TYPE "UDT_ZC_RECETA_CIP_ESTERIL"
VERSION : 0.1
   STRUCT
      TiempoEmpujeADestino : Int;   // ESTERILIZACIÓN. Tiempo de empuje a destino
      TiempoMaxVaciadoDestino : Int;   // ESTERILIZACIÓN. Tiempo Max vaciado destino
      TiempoEmpujeDestinoACIP : Int;   // ESTERILIZACIÓN. Tiempoi empuje desde equipo a CIP
      TiempoMaxEsterilizacion : Int;   // ESTERILIZACIÓN. Tiempo Maximo Enjuague
      TiempoEsterilizacionConConductividad : Int;   // ESTERILIZACIÓN. Tiempo enjuague con conductividad
      ReservaInt_1 : Int;   // ESTERILIZACIÓN.
      ReservaInt_2 : Int;   // ESTERILIZACIÓN.
      TemperaturaEsterilizacion : Real;   // ESTERILIZACIÓN. Temperatura Enjuague
      TemperaturaHisteresis : Real;   // ESTERILIZACIÓN. Temperatura Enjuague Histeresis
      ConductividadDrenaje : Real;   // ESTERILIZACIÓN. Conductividad para Drenaje
      ConductividadEsterilizacion : Real;   // ESTERILIZACIÓN. Conductividad para Enjuague OK
      TemperaturaSalidaEsterilizacion : Real;   // ESTERILIZACIÓN. Temperatura de agua recuperada
      ReservaReal_2 : Real;   // ESTERILIZACIÓN.
   END_STRUCT;

END_TYPE

